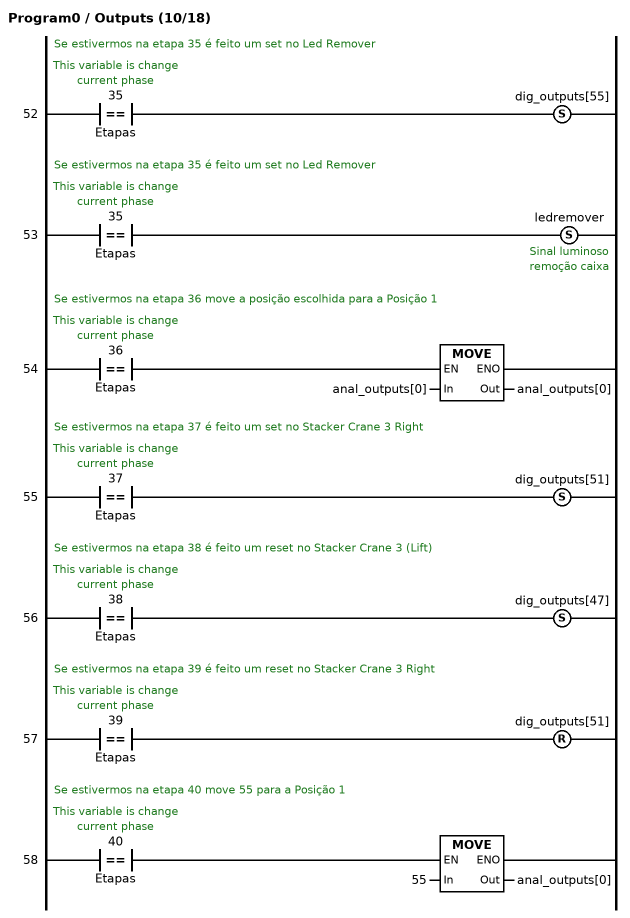
(* [picture p24: Program0 / Outputs, rungs 52-58] *)
(* Rung 52: Se estivermos na etapa 35 é feito um set no Led Remover *)
IF 35 = Etapas THEN dig_outputs[55] := TRUE; END_IF;
(* Rung 53: Se estivermos na etapa 35 é feito um set no Led Remover *)
IF 35 = Etapas THEN ledremover := TRUE; END_IF;
(* Rung 54: Se estivermos na etapa 36 move a posição escolhida para a Posição 1 *)
IF 36 = Etapas THEN anal_outputs[0] := anal_outputs[0]; END_IF;
(* Rung 55: Se estivermos na etapa 37 é feito um set no Stacker Crane 3 Right *)
IF 37 = Etapas THEN dig_outputs[51] := TRUE; END_IF;
(* Rung 56: Se estivermos na etapa 38 é feito um reset no Stacker Crane 3 (Lift) *)
IF 38 = Etapas THEN dig_outputs[47] := TRUE; END_IF;
(* Rung 57: Se estivermos na etapa 39 é feito um reset no Stacker Crane 3 Right *)
IF 39 = Etapas THEN dig_outputs[51] := FALSE; END_IF;
(* Rung 58: Se estivermos na etapa 40 move 55 para a Posição 1 *)
IF 40 = Etapas THEN anal_outputs[0] := 55; END_IF;

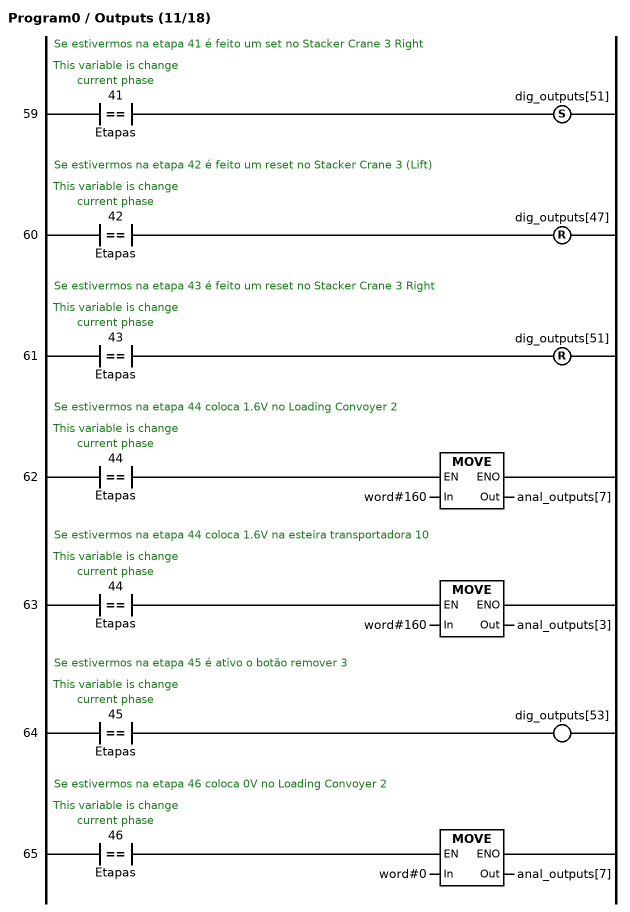
(* Rung 59: Se estivermos na etapa 41 é feito um set no Stacker Crane 3 Right *)
IF 41 = Etapas THEN dig_outputs[51] := TRUE; END_IF;
(* Rung 60: Se estivermos na etapa 42 é feito um reset no Stacker Crane 3 (Lift) *)
IF 42 = Etapas THEN dig_outputs[47] := FALSE; END_IF;
(* Rung 61: Se estivermos na etapa 43 é feito um reset no Stacker Crane 3 Right *)
IF 43 = Etapas THEN dig_outputs[51] := FALSE; END_IF;
(* Rung 62: Se estivermos na etapa 44 coloca 1.6V no Loading Convoyer 2 *)
IF 44 = Etapas THEN anal_outputs[7] := word#160; END_IF;
(* Rung 63: Se estivermos na etapa 44 coloca 1.6V na esteira transportadora 10 *)
IF 44 = Etapas THEN anal_outputs[3] := word#160; END_IF;
(* Rung 64: Se estivermos na etapa 45 é ativo o botão remover 3 *)
dig_outputs[53] := 45 = Etapas;
(* Rung 65: Se estivermos na etapa 46 coloca 0V no Loading Convoyer 2 *)
IF 46 = Etapas THEN anal_outputs[7] := word#0; END_IF;

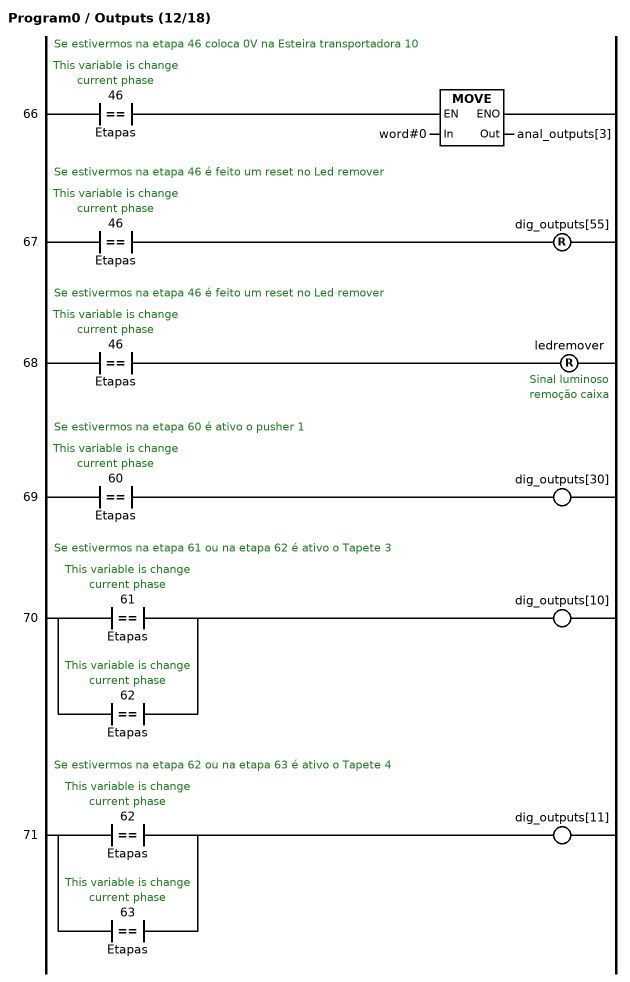
(* Rung 66: Se estivermos na etapa 46 coloca 0V na Esteira transportadora 10 *)
IF 46 = Etapas THEN anal_outputs[3] := word#0; END_IF;
(* Rung 67: Se estivermos na etapa 46 é feito um reset no Led remover *)
IF 46 = Etapas THEN dig_outputs[55] := FALSE; END_IF;
(* Rung 68: Se estivermos na etapa 46 é feito um reset no Led remover *)
IF 46 = Etapas THEN ledremover := FALSE; END_IF;
(* Rung 69: Se estivermos na etapa 60 é ativo o pusher 1 *)
dig_outputs[30] := 60 = Etapas;
(* Rung 70: Se estivermos na etapa 61 ou na etapa 62 é ativo o Tapete 3 *)
dig_outputs[10] := (61 = Etapas) OR (62 = Etapas);
(* Rung 71: Se estivermos na etapa 62 ou na etapa 63 é ativo o Tapete 4 *)
dig_outputs[11] := (62 = Etapas) OR (63 = Etapas);

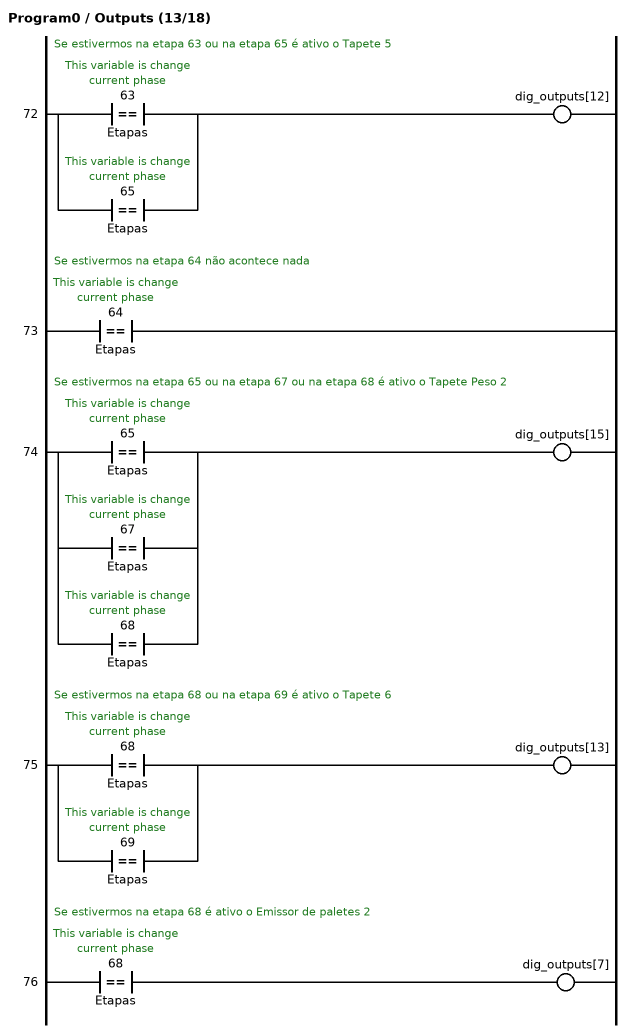
(* Rung 72: Se estivermos na etapa 63 ou na etapa 65 é ativo o Tapete 5 *)
dig_outputs[12] := (63 = Etapas) OR (65 = Etapas);
(* Rung 73: Se estivermos na etapa 64 não acontece nada *)
(* drawn but driving nothing: Etapas *)
(* Rung 74: Se estivermos na etapa 65 ou na etapa 67 ou na etapa 68 é ativo o Tapete Peso 2 *)
dig_outputs[15] := (65 = Etapas) OR (67 = Etapas) OR (68 = Etapas);
(* Rung 75: Se estivermos na etapa 68 ou na etapa 69 é ativo o Tapete 6 *)
dig_outputs[13] := (68 = Etapas) OR (69 = Etapas);
(* Rung 76: Se estivermos na etapa 68 é ativo o Emissor de paletes 2 *)
dig_outputs[7] := 68 = Etapas;

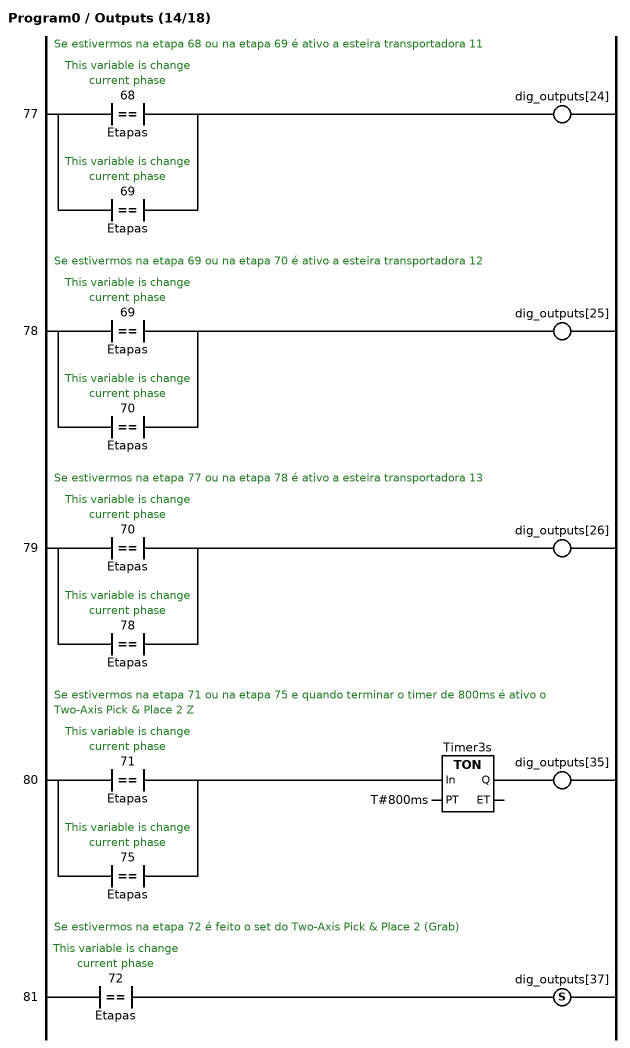
(* Rung 77: Se estivermos na etapa 68 ou na etapa 69 é ativo a esteira transportadora 11 *)
dig_outputs[24] := (68 = Etapas) OR (69 = Etapas);
(* Rung 78: Se estivermos na etapa 69 ou na etapa 70 é ativo a esteira transportadora 12 *)
dig_outputs[25] := (69 = Etapas) OR (70 = Etapas);
(* Rung 79: Se estivermos na etapa 77 ou na etapa 78 é ativo a esteira transportadora 13 *)
dig_outputs[26] := (70 = Etapas) OR (78 = Etapas);
(* Rung 80: Se estivermos na etapa 71 ou na etapa 75 e quando terminar o timer de 800ms é ativo o Two-Axis Pick & Place 2 Z *)
Timer3s(In := (71 = Etapas) OR (75 = Etapas), PT := T#800ms);
dig_outputs[35] := Timer3s.Q;
(* Rung 81: Se estivermos na etapa 72 é feito o set do Two-Axis Pick & Place 2 (Grab) *)
IF 72 = Etapas THEN dig_outputs[37] := TRUE; END_IF;

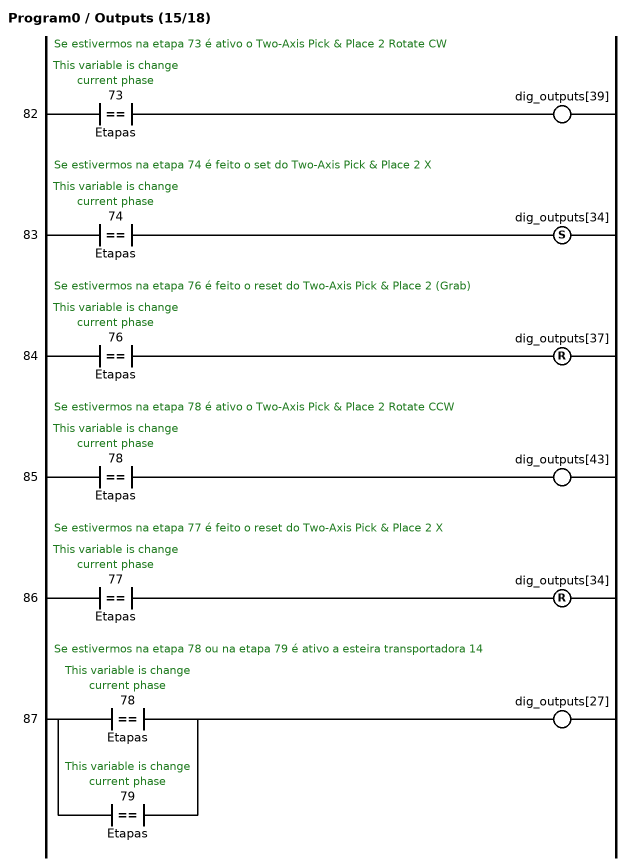
(* Rung 82: Se estivermos na etapa 73 é ativo o Two-Axis Pick & Place 2 Rotate CW *)
dig_outputs[39] := 73 = Etapas;
(* Rung 83: Se estivermos na etapa 74 é feito o set do Two-Axis Pick & Place 2 X *)
IF 74 = Etapas THEN dig_outputs[34] := TRUE; END_IF;
(* Rung 84: Se estivermos na etapa 76 é feito o reset do Two-Axis Pick & Place 2 (Grab) *)
IF 76 = Etapas THEN dig_outputs[37] := FALSE; END_IF;
(* Rung 85: Se estivermos na etapa 78 é ativo o Two-Axis Pick & Place 2 Rotate CCW *)
dig_outputs[43] := 78 = Etapas;
(* Rung 86: Se estivermos na etapa 77 é feito o reset do Two-Axis Pick & Place 2 X *)
IF 77 = Etapas THEN dig_outputs[34] := FALSE; END_IF;
(* Rung 87: Se estivermos na etapa 78 ou na etapa 79 é ativo a esteira transportadora 14 *)
dig_outputs[27] := (78 = Etapas) OR (79 = Etapas);

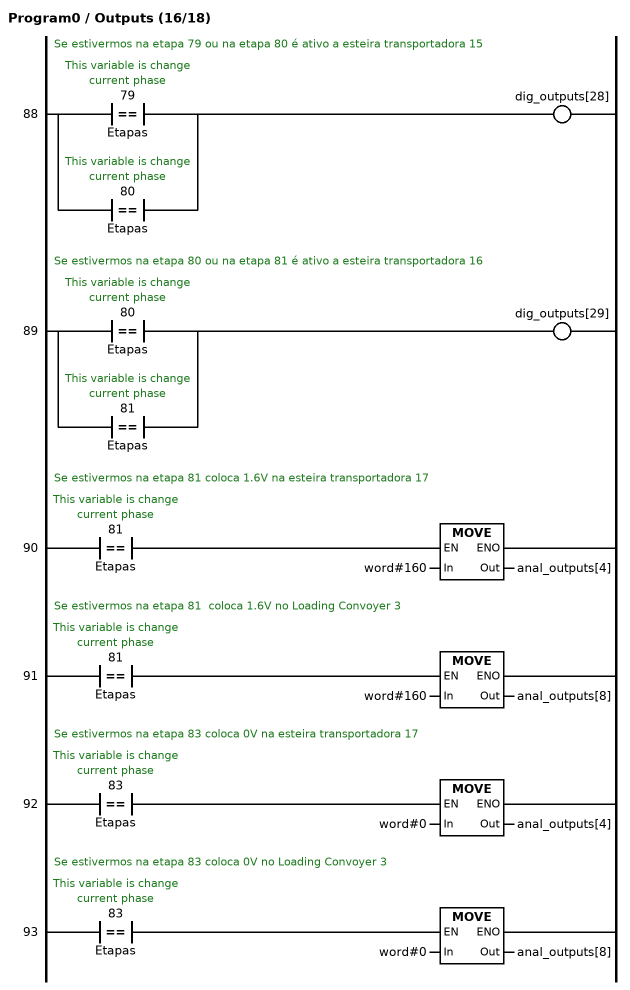
(* Rung 88: Se estivermos na etapa 79 ou na etapa 80 é ativo a esteira transportadora 15 *)
dig_outputs[28] := (79 = Etapas) OR (80 = Etapas);
(* Rung 89: Se estivermos na etapa 80 ou na etapa 81 é ativo a esteira transportadora 16 *)
dig_outputs[29] := (80 = Etapas) OR (81 = Etapas);
(* Rung 90: Se estivermos na etapa 81 coloca 1.6V na esteira transportadora 17 *)
IF 81 = Etapas THEN anal_outputs[4] := word#160; END_IF;
(* Rung 91: Se estivermos na etapa 81  coloca 1.6V no Loading Convoyer 3 *)
IF 81 = Etapas THEN anal_outputs[8] := word#160; END_IF;
(* Rung 92: Se estivermos na etapa 83 coloca 0V na esteira transportadora 17 *)
IF 83 = Etapas THEN anal_outputs[4] := word#0; END_IF;
(* Rung 93: Se estivermos na etapa 83 coloca 0V no Loading Convoyer 3 *)
IF 83 = Etapas THEN anal_outputs[8] := word#0; END_IF;

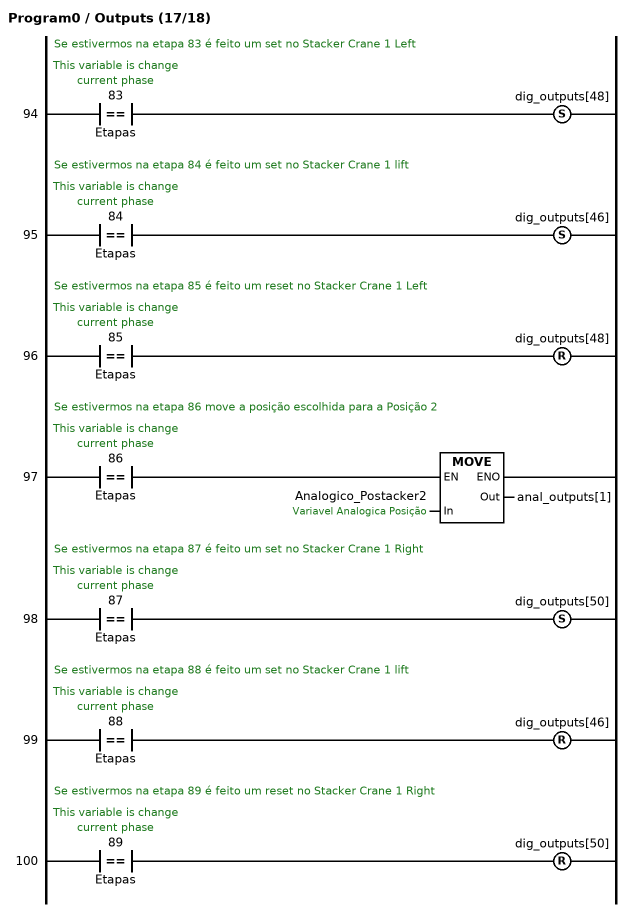
(* Rung 94: Se estivermos na etapa 83 é feito um set no Stacker Crane 1 Left *)
IF 83 = Etapas THEN dig_outputs[48] := TRUE; END_IF;
(* Rung 95: Se estivermos na etapa 84 é feito um set no Stacker Crane 1 lift *)
IF 84 = Etapas THEN dig_outputs[46] := TRUE; END_IF;
(* Rung 96: Se estivermos na etapa 85 é feito um reset no Stacker Crane 1 Left *)
IF 85 = Etapas THEN dig_outputs[48] := FALSE; END_IF;
(* Rung 97: Se estivermos na etapa 86 move a posição escolhida para a Posição 2 *)
IF 86 = Etapas THEN anal_outputs[1] := Analogico_Postacker2; END_IF;
(* Rung 98: Se estivermos na etapa 87 é feito um set no Stacker Crane 1 Right *)
IF 87 = Etapas THEN dig_outputs[50] := TRUE; END_IF;
(* Rung 99: Se estivermos na etapa 88 é feito um set no Stacker Crane 1 lift *)
IF 88 = Etapas THEN dig_outputs[46] := FALSE; END_IF;
(* Rung 100: Se estivermos na etapa 89 é feito um reset no Stacker Crane 1 Right *)
IF 89 = Etapas THEN dig_outputs[50] := FALSE; END_IF;

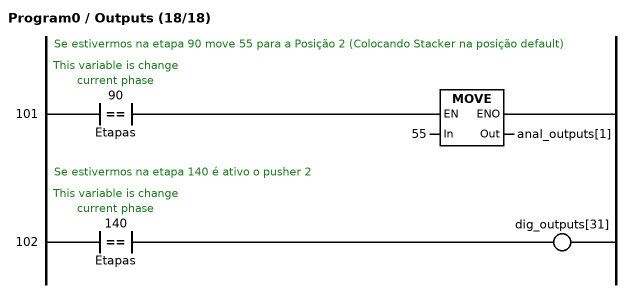
(* Rung 101: Se estivermos na etapa 90 move 55 para a Posição 2 (Colocando Stacker na posição default) *)
IF 90 = Etapas THEN anal_outputs[1] := 55; END_IF;
(* Rung 102: Se estivermos na etapa 140 é ativo o pusher 2 *)
dig_outputs[31] := 140 = Etapas;
END_PROGRAM